{attribute addProperty BoxType "EK1100-0000-0018"}
{attribute addProperty Id "Beckhoff_EL69xxEK1122Beckhoff_EL69xxEK1122_A2B2F2D8162A_0001_EL6900_0000_0016EL6900_4A62393614618.25A_0002_EL6900_0000_0017EL6900_4A62393614618.25A_0003_EL6900_0000_0018EL6900_4A62393614618.25A_0004_EL6900_0000_0019EL6900_4A62393614618.25A_0005_EL6910_0000_0017EL6910_4EA245C69812.25A_0006_EL6910_0000_0018EL6910_4EA245C69812.25A_0007_EL6910_0000_0019EL6910_4EA245C69812.25A_0008_EL6910_0000_0020EL6910_4EA245C69812.25A_0009_EL6930_0000_0016EL6930_4A62393614618.25A_0010_EL6930_0000_0017EL6930_4A62393614618.25A_0011_EL6930_0000_0018EL6930_4A62393614618.25"}
{attribute addProperty CRC "2753439783"}
{attribute addProperty SizeInBites "1430"}
{attribute addProperty SizeInBytes "178.75"}
TYPE Beckhoff_EL69xx_A41E2827 EXTENDS EK1100_179A0949 :
STRUCT
	{attribute addProperty Name "Beckhoff_EL69xxEK1122"}
	Beckhoff_EL69xxEK1122 : Beckhoff_EL69xxEK1122_A2B2F2D8;
	{attribute addProperty Name "A_0001_EL6900_0000_0016"}
	A_0001_EL6900_0000_0016 : EL6900_4A623936;
	{attribute addProperty Name "A_0002_EL6900_0000_0017"}
	A_0002_EL6900_0000_0017 : EL6900_4A623936;
	{attribute addProperty Name "A_0003_EL6900_0000_0018"}
	A_0003_EL6900_0000_0018 : EL6900_4A623936;
	{attribute addProperty Name "A_0004_EL6900_0000_0019"}
	A_0004_EL6900_0000_0019 : EL6900_4A623936;
	{attribute addProperty Name "A_0005_EL6910_0000_0017"}
	A_0005_EL6910_0000_0017 : EL6910_4EA245C6;
	{attribute addProperty Name "A_0006_EL6910_0000_0018"}
	A_0006_EL6910_0000_0018 : EL6910_4EA245C6;
	{attribute addProperty Name "A_0007_EL6910_0000_0019"}
	A_0007_EL6910_0000_0019 : EL6910_4EA245C6;
	{attribute addProperty Name "A_0008_EL6910_0000_0020"}
	A_0008_EL6910_0000_0020 : EL6910_4EA245C6;
	{attribute addProperty Name "A_0009_EL6930_0000_0016"}
	A_0009_EL6930_0000_0016 : EL6930_4A623936;
	{attribute addProperty Name "A_0010_EL6930_0000_0017"}
	A_0010_EL6930_0000_0017 : EL6930_4A623936;
	{attribute addProperty Name "A_0011_EL6930_0000_0018"}
	A_0011_EL6930_0000_0018 : EL6930_4A623936;
END_STRUCT
END_TYPE

(* stored: Version 1.2.0.0, ProductVersion 3.1.4024.9
   DUT Beckhoff_EL69xx_A41E2827: Id {9d8f5a07-22ba-4ce2-9159-089cde9446c1} *)
